// TIA Portal V20 export
VAR_GLOBAL   // PLC tag table "BW_Output"
   AQ_LifeFlag AT %QW500 : Int;
   DQ_LoaderRequest AT %Q502.0 : Bool;
   DQ_LockShuttle AT %Q504.0 : Bool;
   AQ_DataSend AT %QW506 : Int;
   AQ_DataReceive AT %QW508 : Int;
   DQ_NoEmergencyStopAtFemto AT %Q510.0 : Bool;
   DQ_SafetyDoorsClosedAtFemto AT %Q512.0 : Bool;
   AQ_FemtoInErrorState AT %QW514 : Int;
   DQ_AutoMode AT %Q516.0 : Bool;
   DQ_JogMode AT %Q518.0 : Bool;
   DQ_GotoSafePos AT %Q520.0 : Bool;
   AQ_Reset AT %QW526 : Int;
   DQ_Emptying AT %Q522.0 : Bool;
   DQ_BW_CtrlInProgress AT %Q524.0 : Bool;
END_VAR
